// TIA Portal V20 export
DATA_BLOCK "SBK01"   // DB322
// stored: MemoryReserve 100
   VAR
      SPARE : Bool := FALSE;
      "EMO02 CH.A" : Bool := TRUE;
      SPARE_1 : Bool := FALSE;
      "EMO04 CH.A" : Bool := TRUE;
      "EMO01 CH.B" : Bool;
      "EMO02 CH.B" : Bool;
      SPARE_2 : Bool;
      "EMO04 CH.B" : Bool;
      SPARE_3 : Bool;
      SPARE_4 : Bool;
      SPARE_5 : Bool;
   END_VAR
BEGIN
END_DATA_BLOCK
